FUNCTION_BLOCK AxisControl
VAR
	ax			: AXIS_REF;
	mcPower		: MC_Power;
	mcReset		: MC_Reset;
	mcMoveVel	: MC_MoveVelocity;
	mcHalt		: MC_Halt;
	
	_powerOn	: BOOL;
	_reset		: BOOL;
	_moveVel	: BOOL;
	_stop		: BOOL;
	_velocity	: LREAL;
END_VAR

ax.ReadStatus();

mcPower(Axis:= ax, Enable:= _powerOn, Enable_Positive:= _powerOn,	Enable_Negative:= _powerOn);

mcReset(Axis:= ax, Execute:= _reset);
IF mcReset.Done THEN
	mcReset(Axis:= ax, Execute:= FALSE);
	_reset := FALSE;
END_IF

mcMoveVel(Axis:= ax, Execute:= _moveVel, Velocity:= _velocity);
IF mcMoveVel.InVelocity THEN
	_moveVel := FALSE;
END_IF

mcHalt(Axis:= ax, Execute:= _stop);	
IF mcHalt.Done THEN
	_stop := FALSE;
END_IF

PROPERTY AxisError : DWORD
GET
AxisError := UDINT_TO_DWORD(ax.Status.ErrorID);
END_GET
END_PROPERTY

METHOD MoveAxis : BOOL
VAR_INPUT
	Velocity: LREAL := 0.1;
END_VAR
_moveVel := TRUE;
_stop := FALSE;
_velocity := Velocity;

MoveAxis := TRUE;
END_METHOD

PROPERTY Position : LREAL
GET
Position := ax.NcToPlc.ActPos;
END_GET
END_PROPERTY

METHOD PowerAxis : BOOL
VAR_INPUT
	Enable: BOOL;
END_VAR
_powerOn := Enable;

PowerAxis := TRUE;
END_METHOD

METHOD Reset : BOOL
_reset := TRUE;
_moveVel := FALSE;
_stop := FALSE;

Reset := TRUE;
END_METHOD

METHOD StopAxis : BOOL
_moveVel := FALSE;
_stop := TRUE;

StopAxis := TRUE;
END_METHOD

END_FUNCTION_BLOCK

(* stored: Version 1.1.0.1, ProductVersion 3.1.4026.18
   POU AxisControl: Id {57c58ad5-0d08-07cf-1746-26196577400b}, SpecialFunc None
   Property AxisError: Id {e84503b5-93a8-0859-271c-b99c5ca74dd1}
   Get Get: Id {9495b105-4825-055a-0565-394aaa01e9a5}
   Method MoveAxis: Id {2ed2d19d-343b-025d-2400-9ce26d08a296}
   Property Position: Id {01aeaff8-1d4a-0112-0c1e-49d99f9bafa7}
   Get Get: Id {bff4513a-6377-0d14-3a21-e4ad17db4400}
   Method PowerAxis: Id {0df46747-2c5a-0e25-1098-6a7255e56a86}
   Method Reset: Id {979dfdb8-d934-02cf-1fda-32b040f4c3d4}
   Method StopAxis: Id {0bb9adb9-2e2c-03fc-31c7-504b2b35be51} *)
